# EPICS substitutions: db/el3164.substitutions
file el3164.template
{
	pattern {CH_ID, PDO_IDX}
		{$(MOD_ID)-AI1, 0}
		{$(MOD_ID)-AI2, 1}
		{$(MOD_ID)-AI3, 2}
		{$(MOD_ID)-AI4, 3}
}
